// SIMATIC STEP 7 (V5.x) project PROBLEM 9
// CPU: CPU 314C-2 DP
// station: Hardware
// station: SIMATIC 300(1)
// station: P_ADR_BUS
// program: S7 Program(1)

ORGANIZATION_BLOCK OB 1
TITLE = "Main Program Sweep (Cycle)"
VERSION : 0.1
VAR_TEMP
  OB1_EV_CLASS : BYTE ;	//Bits 0-3 = 1 (Coming event), Bits 4-7 = 1 (Event class 1)
  OB1_SCAN_1 : BYTE ;	//1 (Cold restart scan 1 of OB 1), 3 (Scan 2-n of OB 1)
  OB1_PRIORITY : BYTE ;	//Priority of OB Execution
  OB1_OB_NUMBR : BYTE ;	//1 (Organization block 1, OB1)
  OB1_RESERVED_1 : BYTE ;	//Reserved for system
  OB1_RESERVED_2 : BYTE ;	//Reserved for system
  OB1_PREV_CYCLE : INT ;	//Cycle time of previous OB1 scan (milliseconds)
  OB1_MIN_CYCLE : INT ;	//Minimum cycle time of OB1 (milliseconds)
  OB1_MAX_CYCLE : INT ;	//Maximum cycle time of OB1 (milliseconds)
  OB1_DATE_TIME : DATE_AND_TIME ;	//Date and time OB1 started
END_VAR
BEGIN
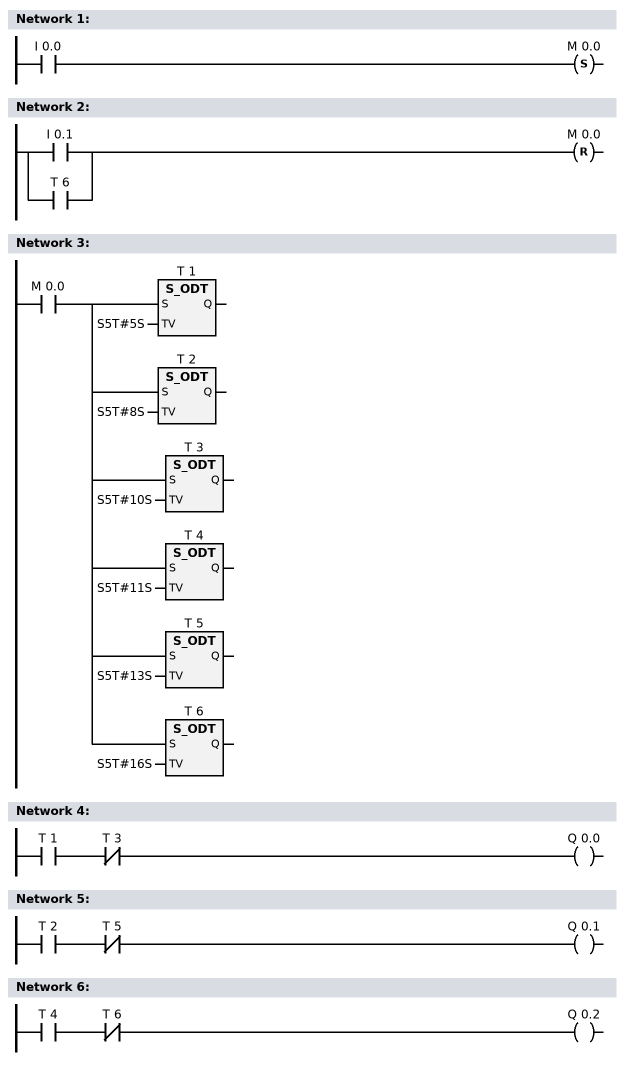
NETWORK
TITLE =
      A     I 0.0;
      S     M 0.0;
NETWORK
TITLE =
      O     I 0.1;
      O     T 6;
      R     M 0.0;
NETWORK
TITLE =
      A     M 0.0;
      =     L 20.0;
      A     L 20.0;
      L     S5T#5S;
      SD    T 1;
      NOP   0;
      NOP   0;
      NOP   0;
      NOP   0;
      A     L 20.0;
      L     S5T#8S;
      SD    T 2;
      NOP   0;
      NOP   0;
      NOP   0;
      NOP   0;
      A     L 20.0;
      L     S5T#10S;
      SD    T 3;
      NOP   0;
      NOP   0;
      NOP   0;
      NOP   0;
      A     L 20.0;
      L     S5T#11S;
      SD    T 4;
      NOP   0;
      NOP   0;
      NOP   0;
      NOP   0;
      A     L 20.0;
      L     S5T#13S;
      SD    T 5;
      NOP   0;
      NOP   0;
      NOP   0;
      NOP   0;
      A     L 20.0;
      L     S5T#16S;
      SD    T 6;
      NOP   0;
      NOP   0;
      NOP   0;
      NOP   0;
NETWORK
TITLE =
      A     T 1;
      AN    T 3;
      =     Q 0.0;
NETWORK
TITLE =
      A     T 2;
      AN    T 5;
      =     Q 0.1;
NETWORK
TITLE =
      A     T 4;
      AN    T 6;
      =     Q 0.2;
END_ORGANIZATION_BLOCK
